TYPE eFiltertyp :
(
	NONE_ := 1,
	TIEFPASS := 2,
	HOCHPASS := 3
);
END_TYPE

(* stored: Version 1.1.0.1, ProductVersion 3.1.4024.12
   DUT eFiltertyp: Id {44d1ec65-7fd9-45d9-a612-819cb16c8945} *)
